TYPE MC_COMMAND_REF :
STRUCT
	CommandId: INT;
END_STRUCT
END_TYPE

(* stored: Version 1.1.0.1, ProductVersion 3.1.4024.11
   DUT MC_COMMAND_REF: Id {e9f505d9-c431-4cec-bc71-df5ca88a0cc0} *)
